{attribute 'GeneratedUsingTerminal: EJ2521-0224-0016'}
{attribute addProperty BoxType "EJ2521-0224-0016"}
{attribute addProperty Id "StatusAT %I*Status_7097155E4"}
{attribute addProperty CRC "1894228450"}
{attribute addProperty Size "4"}
TYPE PLS_Status_Channel_70E7A1E2 :
STRUCT
	{attribute addProperty Name "Status"}
	Status AT %I* : Status_7097155E;
END_STRUCT
END_TYPE
